{attribute 'GeneratedUsingTerminal: EK1100-0000-0018'}
{attribute addProperty BoxType "EK1100-0000-0018"}
{attribute addProperty Id "Beckhoff_EL37xxEK1122Beckhoff_EL37xxEK1122_217FAF052A_0001_EL3702_0000_0002EL3702_C321C59156A_0002_EL3702_0000_0003EL3702_C321C59156A_0003_EL3702_0015_0003EL3702_C321C59156A_0004_EL3742_0000_0001EL3742_30F92DF722A_0005_EL3742_0000_0002EL3742_C321C59156A_0006_EL3742_0000_0003EL3742_C321C59156A_0007_EL3751_0000_0020EL3751_0538829531A_0008_EL3751_0000_0021EL3751_0538829531A_0009_EL3751_0000_0022EL3751_0538829531A_0010_EL3751_0000_0023EL3751_0538829531A_0011_EL3751_0004_0022EL3751_0538829531A_0012_EL3751_0004_0023EL3751_0538829531A_0013_EL3751_0020_0020EL3751_0538829531A_0014_EL3751_0020_0021EL3751_0538829531A_0015_EL3751_0020_0022EL3751_0538829531A_0016_EL3751_0020_0023EL3751_0538829531A_0017_EL3751_0024_0022EL3751_0538829531A_0018_EL3751_0024_0023EL3751_0538829531A_0019_EL3773_0000_0016EL3773_598F0172190A_0020_EL3773_0000_0017EL3773_B0EE24E7190A_0021_EL3773_0000_0018EL3773_E277286D184A_0022_EL3773_0000_0019EL3773_DA71AF99184A_0023_EL3773_0000_0020EL3773_DA71AF99184A_0024_EL3773_0000_0021EL3773_DA71AF99184A_0025_EL3783_0000_0018EL3783_DD6F4D3B309"}
{attribute addProperty CRC "4196355125"}
{attribute addProperty Size "2101"}
TYPE Beckhoff_EL37xx_FA1F4C35 EXTENDS EK1100_1FC0878B :
STRUCT
	{attribute addProperty Name "Beckhoff_EL37xxEK1122"}
	{attribute addProperty PreviousPort "Beckhoff EL37xx : B"}
	Beckhoff_EL37xxEK1122 : Beckhoff_EL37xxEK1122_217FAF05;
	{attribute addProperty Name "A_0001_EL3702_0000_0002"}
	{attribute addProperty PreviousPort "Beckhoff EL37xxEK1122 : C"}
	A_0001_EL3702_0000_0002 : EL3702_C321C591;
	{attribute addProperty Name "A_0002_EL3702_0000_0003"}
	{attribute addProperty PreviousPort "A_0001(EL3702-0000-0002) : B"}
	A_0002_EL3702_0000_0003 : EL3702_C321C591;
	{attribute addProperty Name "A_0003_EL3702_0015_0003"}
	{attribute addProperty PreviousPort "A_0002(EL3702-0000-0003) : B"}
	A_0003_EL3702_0015_0003 : EL3702_C321C591;
	{attribute addProperty Name "A_0004_EL3742_0000_0001"}
	{attribute addProperty PreviousPort "A_0003(EL3702-0015-0003) : B"}
	A_0004_EL3742_0000_0001 : EL3742_30F92DF7;
	{attribute addProperty Name "A_0005_EL3742_0000_0002"}
	{attribute addProperty PreviousPort "A_0004(EL3742-0000-0001) : B"}
	A_0005_EL3742_0000_0002 : EL3742_C321C591;
	{attribute addProperty Name "A_0006_EL3742_0000_0003"}
	{attribute addProperty PreviousPort "A_0005(EL3742-0000-0002) : B"}
	A_0006_EL3742_0000_0003 : EL3742_C321C591;
	{attribute addProperty Name "A_0007_EL3751_0000_0020"}
	{attribute addProperty PreviousPort "A_0006(EL3742-0000-0003) : B"}
	A_0007_EL3751_0000_0020 : EL3751_05388295;
	{attribute addProperty Name "A_0008_EL3751_0000_0021"}
	{attribute addProperty PreviousPort "A_0007(EL3751-0000-0020) : B"}
	A_0008_EL3751_0000_0021 : EL3751_05388295;
	{attribute addProperty Name "A_0009_EL3751_0000_0022"}
	{attribute addProperty PreviousPort "A_0008(EL3751-0000-0021) : B"}
	A_0009_EL3751_0000_0022 : EL3751_05388295;
	{attribute addProperty Name "A_0010_EL3751_0000_0023"}
	{attribute addProperty PreviousPort "A_0009(EL3751-0000-0022) : B"}
	A_0010_EL3751_0000_0023 : EL3751_05388295;
	{attribute addProperty Name "A_0011_EL3751_0004_0022"}
	{attribute addProperty PreviousPort "A_0010(EL3751-0000-0023) : B"}
	A_0011_EL3751_0004_0022 : EL3751_05388295;
	{attribute addProperty Name "A_0012_EL3751_0004_0023"}
	{attribute addProperty PreviousPort "A_0011(EL3751-0004-0022) : B"}
	A_0012_EL3751_0004_0023 : EL3751_05388295;
	{attribute addProperty Name "A_0013_EL3751_0020_0020"}
	{attribute addProperty PreviousPort "A_0012(EL3751-0004-0023) : B"}
	A_0013_EL3751_0020_0020 : EL3751_05388295;
	{attribute addProperty Name "A_0014_EL3751_0020_0021"}
	{attribute addProperty PreviousPort "A_0013(EL3751-0020-0020) : B"}
	A_0014_EL3751_0020_0021 : EL3751_05388295;
	{attribute addProperty Name "A_0015_EL3751_0020_0022"}
	{attribute addProperty PreviousPort "A_0014(EL3751-0020-0021) : B"}
	A_0015_EL3751_0020_0022 : EL3751_05388295;
	{attribute addProperty Name "A_0016_EL3751_0020_0023"}
	{attribute addProperty PreviousPort "A_0015(EL3751-0020-0022) : B"}
	A_0016_EL3751_0020_0023 : EL3751_05388295;
	{attribute addProperty Name "A_0017_EL3751_0024_0022"}
	{attribute addProperty PreviousPort "A_0016(EL3751-0020-0023) : B"}
	A_0017_EL3751_0024_0022 : EL3751_05388295;
	{attribute addProperty Name "A_0018_EL3751_0024_0023"}
	{attribute addProperty PreviousPort "A_0017(EL3751-0024-0022) : B"}
	A_0018_EL3751_0024_0023 : EL3751_05388295;
	{attribute addProperty Name "A_0019_EL3773_0000_0016"}
	{attribute addProperty PreviousPort "A_0018(EL3751-0024-0023) : B"}
	A_0019_EL3773_0000_0016 : EL3773_598F0172;
	{attribute addProperty Name "A_0020_EL3773_0000_0017"}
	{attribute addProperty PreviousPort "A_0019(EL3773-0000-0016) : B"}
	A_0020_EL3773_0000_0017 : EL3773_B0EE24E7;
	{attribute addProperty Name "A_0021_EL3773_0000_0018"}
	{attribute addProperty PreviousPort "A_0020(EL3773-0000-0017) : B"}
	A_0021_EL3773_0000_0018 : EL3773_E277286D;
	{attribute addProperty Name "A_0022_EL3773_0000_0019"}
	{attribute addProperty PreviousPort "A_0021(EL3773-0000-0018) : B"}
	A_0022_EL3773_0000_0019 : EL3773_DA71AF99;
	{attribute addProperty Name "A_0023_EL3773_0000_0020"}
	{attribute addProperty PreviousPort "A_0022(EL3773-0000-0019) : B"}
	A_0023_EL3773_0000_0020 : EL3773_DA71AF99;
	{attribute addProperty Name "A_0024_EL3773_0000_0021"}
	{attribute addProperty PreviousPort "A_0023(EL3773-0000-0020) : B"}
	A_0024_EL3773_0000_0021 : EL3773_DA71AF99;
	{attribute addProperty Name "A_0025_EL3783_0000_0018"}
	{attribute addProperty PreviousPort "A_0024(EL3773-0000-0021) : B"}
	A_0025_EL3783_0000_0018 : EL3783_DD6F4D3B;
END_STRUCT
END_TYPE

(* stored: Version 1.2.0.0, ProductVersion 3.1.4024.9
   DUT Beckhoff_EL37xx_FA1F4C35: Id {084242bf-1d17-4978-8f9b-4d1589d64dbe} *)
